{attribute 'qualified_only'}
VAR_GLOBAL
	Status						:	BOOL	;
	NO							:	INT		;
	Wait_Vision					: 	BOOL	;
	Data_Copy					:	BOOL	;
	Vision_Data_Apply			: 	BOOL	;
	Wait_Start_Sensor			: 	BOOL	;
	Moving_Start				: 	BOOL	;
	Axis04_Comp					: 	BOOL	;
	Axis04_Work_Comp			: 	BOOL	;
	Axis04_Work_Comp_Wait		: 	BOOL	;
	Press_5ms					: 	BOOL	;
	Press_Stop					:	BOOL	;
	Axis04_Wait_Pos_Moving		: 	BOOL	;
	Axis02_Work_Comp_Wait		: 	BOOL	;
	Axis02_Wait_Pos_Moving		: 	BOOL	;
	All_Motor_Wait_Pos_Moving	:	BOOL	;
	Vision_Data_Reset			:	BOOL	;
	Vision_Data_Initial			:	BOOL	;
	All_Initial					:	BOOL	;
	Target_Position_Moving		:	BOOL	;
	Press_Start					:	BOOL	;
	Press_Wait					:	BOOL	;
	Axis04_Work_move			:	BOOL	;
	

	Data_Copy_Comp				:	BOOL	;
END_VAR

(* stored: Version 1.1.0.1, ProductVersion 3.1.4024.15
   GVL GVL_Main_Step: Id {4f8bf6f9-b9e8-4d38-a767-00aa9781ac1d} *)
